FUNCTION_BLOCK F_WORD_TO_REAL (* convert WORD to REAL *)
  (* Standard: 61131-3; Classification: standard type conversion function; Description: Copyright (c) 2012 TU Wien ACIN This program and the accompanying materials are made available under the terms of the Eclipse Public License 2.0 which is available at https://www.eclipse.org/legal/epl-2.0/ SPDX-License-Identifier: EPL-2.0 *)
  (* Version 1.0, 2012-01-19, Monika Wenger, TU Wien ACIN *)
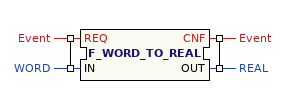
  EVENT_INPUT
    REQ WITH IN; (* Service Request *)
  END_EVENT
  EVENT_OUTPUT
    CNF WITH OUT; (* Confirmation of Requested Service *)
  END_EVENT
  VAR_INPUT
    IN : WORD; (* Event Input Qualifier *)
  END_VAR
  VAR_OUTPUT
    OUT : REAL; (* Event Output Qualifier *)
  END_VAR
END_FUNCTION_BLOCK
